Staubli VAL3: stop.pgx

program stop()
begin
  //库结束
  title("")
  cls()


end
